FUNCTION_BLOCK FB_WindTurbineSim
VAR_INPUT
	windSpeed		: LREAL;
	
END_VAR
VAR_OUTPUT
	rpm				: LREAL;
	powerOutput		: LREAL;
END_VAR
VAR
	risingCoef		: LREAL := 0.000314; //Coefficient for the rising segment for SD6+
	tipSpeed		: LREAL;
	cutInSpeed		: LREAL := 5.59234;	//mph
	
END_VAR

VAR CONSTANT
	radius			: LREAL := 2.8;		//5.6m diameter of SD Wind SD6+ turbine
	tsr				: Lreal	:= 2.5;		//tip speed ration usually arownd 7 for commercial turbines
	maxRPM			: LREAL	:= 200.0;
	maxOperationalSpeed: LREAL := 156.586;	//mph
	ratedSpeed		: LREAL := 30;			//mph
END_VAR

IF windSpeed < 6.00 THEN
	powerOutput := 0.00;
ELSIF windSpeed <= 30.00 THEN
	powerOutput := risingCoef * EXPT(windSpeed, 3);
ELSIF windSpeed <= 55.00 THEN
	powerOutput := 8.5;
ELSE
	powerOutput := 0;
END_IF

IF windSpeed < cutInSpeed THEN
	rpm := 0;
END_IF

IF windSpeed <= ratedSpeed THEN
	tipSpeed := tsr * windSpeed;
	rpm := (tipSpeed * 60) / (3.14 * 2 * radius);
	rpm := MIN(rpm, maxRPM);

ELSE
	rpm := maxRPM;
END_IF

//tipSpeed := tsr * MIN(windSpeed,maxOperationalSpeed);



//IF rpm > maxRPM THEN
//	rpm := maxRPM;
//END_IF

END_FUNCTION_BLOCK

(* stored: Version 1.1.0.1, ProductVersion 3.1.4024.12
   POU FB_WindTurbineSim: Id {094f154f-e176-415b-a9da-91bd88f15827}, SpecialFunc None *)
